# EPICS substitutions: apps/A6551App/Db/original/user.substitutions
# Example substitutions file

file "db/dbExample1.db" {
    { user = "baltzell" }
}

file db/dbExample2.db {
    pattern { user, no, scan }
        { "baltzell", 1, "1 second" }
        { "baltzell", 2, "2 second" }
        { "baltzell", 3, "5 second" }
}
